FUNCTION_BLOCK Display (* Basic FB with empty ECC *)
  (* Standard: 61499-2 *)
  (* Version 1.0, 2022-01-09, Fan *)
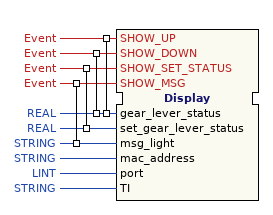
  EVENT_INPUT
    SHOW_UP WITH gear_lever_status;
    SHOW_DOWN WITH gear_lever_status;
    SHOW_SET_STATUS WITH set_gear_lever_status;
    SHOW_MSG WITH msg_light;
  END_EVENT
  VAR_INPUT
    gear_lever_status : REAL;
    set_gear_lever_status : REAL;
    msg_light : STRING;
    mac_address : STRING;
    port : LINT;
    TI : STRING;
  END_VAR
  EC_STATES
    START; (* Initial State *)
  END_STATES
END_FUNCTION_BLOCK
